PROGRAM P_LubLogic
VAR
	TON_MaqLigada 			: TON;
	bMaquinaLigada			: BOOL;
	tEsperaLubrificacao		: TIME := T#30S;
	tLubrificacao			: TIME := T#5S;
	TON_Lubrificando		: TON;
	bFirstScan				: BOOL := TRUE;
	doLubrificacao			: BOOL;
	tiSoma					: TIME;	
	tiSomaOdometro			: TIME;	
END_VAR

VAR PERSISTENT	
	tiOdometro				: TIME;
	tiOdometro_Old			: TIME;
END_VAR
VAR // added by the converter: edge detectors and wires of the graphical bodies
    _w1 : BOOL;
END_VAR

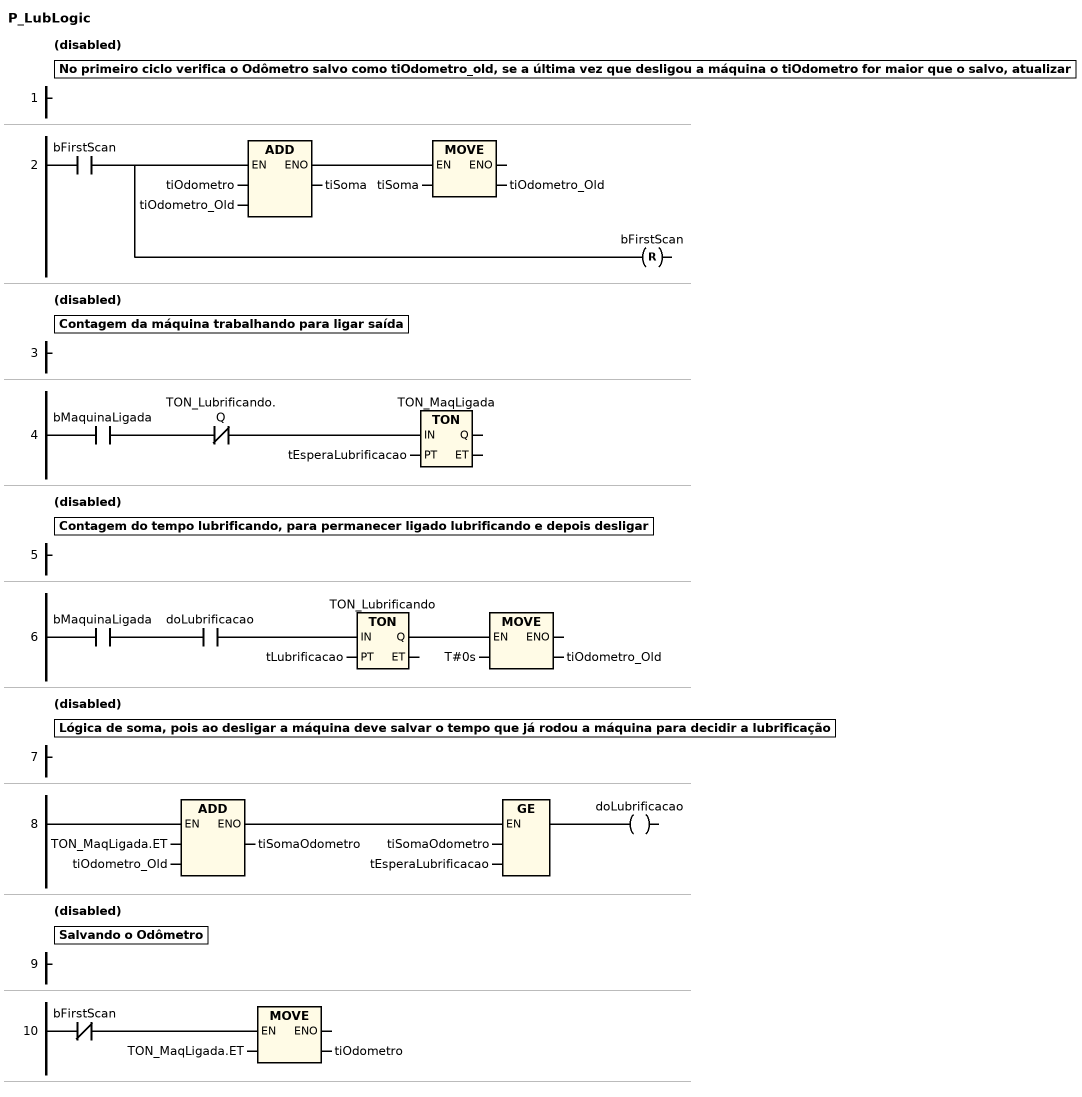
// NETWORK 1 (disabled)
// label: No primeiro ciclo verifica o Odômetro salvo como tiOdometro_old, se a última vez que desligou a máquina o tiOdometro for maior que o salvo, atualizar

// NETWORK 2
_w1 := bFirstScan;
IF _w1 THEN tiSoma := tiOdometro + tiOdometro_Old; END_IF
IF _w1 THEN tiOdometro_Old := tiSoma; END_IF
bFirstScan R= _w1;

// NETWORK 3 (disabled)
// label: Contagem da máquina trabalhando para ligar saída

// NETWORK 4
TON_MaqLigada(IN := bMaquinaLigada AND NOT TON_Lubrificando.Q, PT := tEsperaLubrificacao); // TON

// NETWORK 5 (disabled)
// label: Contagem do tempo lubrificando, para permanecer ligado lubrificando e depois desligar

// NETWORK 6
TON_Lubrificando(IN := bMaquinaLigada AND doLubrificacao, PT := tLubrificacao); // TON
IF TON_Lubrificando.Q THEN tiOdometro_Old := T#0s; END_IF

// NETWORK 7 (disabled)
// label: Lógica de soma, pois ao desligar a máquina deve salvar o tempo que já rodou a máquina para decidir a lubrificação

// NETWORK 8
tiSomaOdometro := TON_MaqLigada.ET + tiOdometro_Old;
doLubrificacao := tiSomaOdometro >= tEsperaLubrificacao;

// NETWORK 9 (disabled)
// label: Salvando o Odômetro

// NETWORK 10
IF NOT bFirstScan THEN tiOdometro := TON_MaqLigada.ET; END_IF

END_PROGRAM

(* stored: Version 1.1.0.1, ProductVersion 3.1.4024.12
   POU P_LubLogic: Id {8dec4306-4789-49f2-94a6-cfbbe0b07868}, SpecialFunc None *)
